PROGRAM MAIN
VAR
	Enable_Axis1: BOOL;
	Enable_Axis2: BOOL;
	Move_Axis1 : BOOL;
	Move_Axis2 : BOOL;
	Abilita_Axis1 : MC_Power;
	Abilita_Axis2 : MC_Power;
	Muovi_Axis1 : MC_MoveRelative;
	Muovi_Axis2 : MC_MoveRelative;
END_VAR

Abilita_Assi();
Muovi_Assi();

ACTION Abilita_Assi:
Abilita_Axis1(
	Axis:= GVL.Axis1, 
	Enable:= Enable_Axis1, 
	Enable_Positive:= TRUE, 
	Enable_Negative:= TRUE, 
	Override:= 100);

Abilita_Axis2(
	Axis:= GVL.Axis2, 
	Enable:= Enable_Axis2, 
	Enable_Positive:= TRUE, 
	Enable_Negative:= TRUE, 
	Override:= 100);
END_ACTION

ACTION Muovi_Assi:
Muovi_Axis1(
	Axis:= GVL.Axis1, 
	Execute:= Move_Axis1, 
	Distance:= 3600, 
	Velocity:= 9000 );
	
Muovi_Axis1(
	Axis:= GVL.Axis2, 
	Execute:= Move_Axis2, 
	Distance:= 3600, 
	Velocity:= 9000 );
END_ACTION

END_PROGRAM

(* stored: Version 1.1.0.1, ProductVersion 3.1.4024.12
   POU MAIN: Id {3bfc9037-5bfd-455d-a6fb-465065dbe6e5}, SpecialFunc None
   Action Abilita_Assi: Id {aa482131-6bed-4b0b-b110-03855a53b825}
   Action Muovi_Assi: Id {f18f75f2-ef74-4fa5-9fa2-5513e7a87f91} *)
